ABB RobotStudio station: Session5.rspag

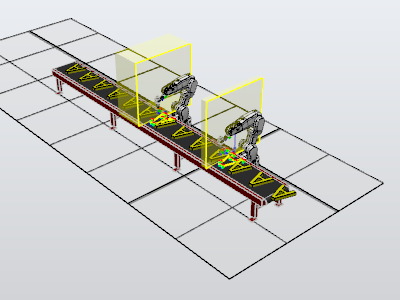
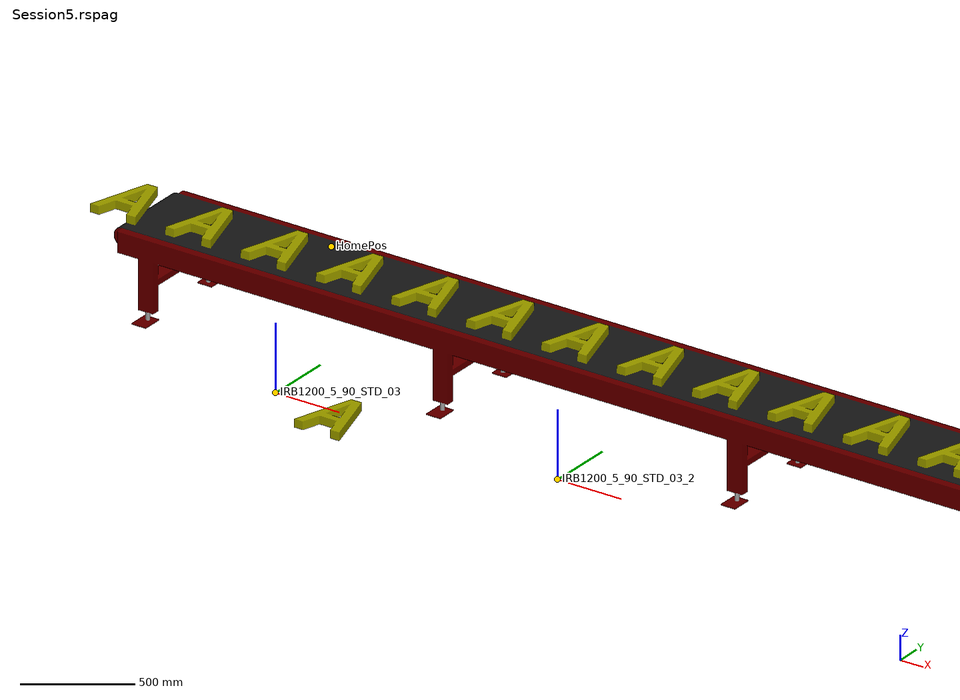
[picture v1: parts stored in the station drawn from their meshes, with robot base, taught points and paths (robot models come from the ABB library and are not in the file)]
--- station ---
Station Session5 (saved by RobotStudio 24.2.10821.1)
Controller IRB1200_CNV_2, task T_ROB1: task frame (RAPID world) sits at (1000, 521.42, 400) mm in the station
Controller IRB1200_CNV_1, task T_ROB1: task frame (RAPID world) sits at (-500, 521.42, 400) mm in the station
Controller IRB1200_CNV_1
  mechanical unit ROB_1: IRB1200_5_90_STD_03, 6 joints, base frame (0, -290, -400) mm, rotated rx 0 ry 0 rz 90 deg
  mechanical unit CNV1: ?, 1 joints, base frame (0, 0, 0) mm
Controller IRB1200_CNV_2
  mechanical unit ROB_1: IRB1200_5_90_STD_03_2, 6 joints, base frame (0, -290, -400) mm, rotated rx 0 ry 0 rz 90 deg
  mechanical unit CNV1: ?, 1 joints, base frame (0, 0, 0) mm
Layout (positions relative to the parent item):
  - IRB1200_5_90_STD_03 [mechanism, from %ABB.RobotStudio.Models.IRB1200%\IRB1200_5_90_STD_03.rslib] at (-500, 231.42, 0) mm, rotated rx 0 ry 0 rz 90 deg; joint values [-0.0648, -0.2584, 0.4127, -0.0339, 0.7666, 0.0529] (rad or m)
  - mySpintecTool [mechanism, from Library\mySpintecTool.rslib] at (-472.99, 617.74, 739.17) mm, rotated rx -179.89 ry 37.27 rz -95.76 deg
  - Conveyor 1 [conveyor]
    - Belt Conveyor [part] at (-518.08, 731.42, 0) mm, size 5091 x 600 x 400 mm
    - Product_A [part], size 239 x 301.5 x 40 mm
    - ConveyorObject_82 [conveyorobject] at (3315.13, 521.42, 400) mm
      - Product_A [part] at (0, 50, 0) mm, size 239 x 301.5 x 40 mm
    - ConveyorObject_83 [conveyorobject] at (2915.13, 521.42, 400) mm
      - Product_A [part] at (0, 50, 0) mm, size 239 x 301.5 x 40 mm
    - ConveyorObject_84 [conveyorobject] at (2515.13, 521.42, 400) mm
      - Product_A [part] at (0, 50, 0) mm, size 239 x 301.5 x 40 mm
    - ConveyorObject_85 [conveyorobject] at (2115.13, 521.42, 400) mm
      - Product_A [part] at (0, 50, 0) mm, size 239 x 301.5 x 40 mm
    - ConveyorObject_86 [conveyorobject] at (1715.13, 521.42, 400) mm
      - Product_A [part] at (0, 50, 0) mm, size 239 x 301.5 x 40 mm
    - ConveyorObject_87 [conveyorobject] at (1315.13, 521.42, 400) mm
      - Product_A [part] at (0, 50, 0) mm, size 239 x 301.5 x 40 mm
    - ConveyorObject_88 [conveyorobject] at (915.13, 521.42, 400) mm
      - Product_A [part] at (0, 50, 0) mm, size 239 x 301.5 x 40 mm
    - ConveyorObject_89 [conveyorobject] at (515.13, 521.42, 400) mm
      - Product_A [part] at (0, 50, 0) mm, size 239 x 301.5 x 40 mm
    - ConveyorObject_90 [conveyorobject] at (115.13, 521.42, 400) mm
      - Product_A [part] at (0, 50, 0) mm, size 239 x 301.5 x 40 mm
    - ConveyorObject_91 [conveyorobject] at (-284.87, 521.42, 400) mm
      - Product_A [part] at (0, 50, 0) mm, size 239 x 301.5 x 40 mm
    - ConveyorObject_92 [conveyorobject] at (-684.87, 521.42, 400) mm
      - Product_A [part] at (0, 50, 0) mm, size 239 x 301.5 x 40 mm
    - ConveyorObject_93 [conveyorobject] at (-1084.87, 521.42, 400) mm
      - Product_A [part] at (0, 50, 0) mm, size 239 x 301.5 x 40 mm
    - ConveyorObject_94 [conveyorobject] at (-1484.87, 521.42, 400) mm
      - Product_A [part] at (0, 50, 0) mm, size 239 x 301.5 x 40 mm
  - IRB1200_5_90_STD_03_2 [mechanism, from %ABB.RobotStudio.Models.IRB1200%\IRB1200_5_90_STD_03.rslib] at (1000, 231.42, 0) mm, rotated rx 0 ry 0 rz 90 deg; joint values [0, -0.4363, 0.5236, 0, 0.8378, 0] (rad or m)
  - mySpintecTool_2 [mechanism, from Library\mySpintecTool.rslib] at (1000, 544.38, 742.17) mm, rotated rx 180 ry 37 rz -90 deg
Attachment: mySpintecTool is attached to IRB1200_5_90_STD_03 / Link6
Attachment: mySpintecTool_2 is attached to IRB1200_5_90_STD_03_2 / Link6
Conveyor tracking Connection: unit CNV1, TravelOffset=1.018075, QueueTrackDistance=0, StartWindowWidth=0.1, SyncSeparation=5E-06, CountsPerMeter=20000
Conveyor tracking Connection_2: unit CNV1, TravelOffset=2.518075, QueueTrackDistance=0, StartWindowWidth=0.5, SyncSeparation=5E-06, CountsPerMeter=20000
Targets, tools, work objects and paths stored in the station and not in the controller backup, written as RAPID:
! task T_ROB1
MODULE Module1
  CONST robtarget Target_10:=[[0,50,40],[0,-0.595435711,0.803402959,0],[0,0,0,0],[9E+09,9E+09,9E+09,9E+09,9E+09,0]];
ENDMODULE


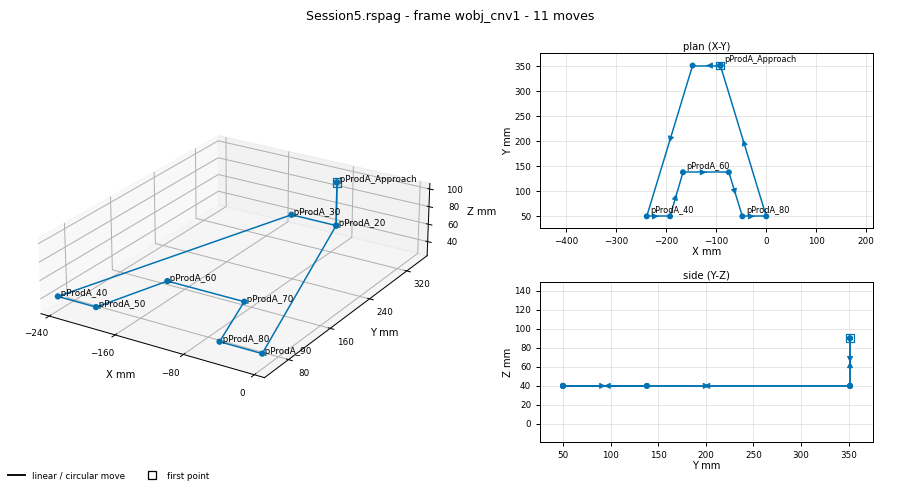
[picture p0: tool path of Session5.rspag in frame wobj_cnv1, 11 of 13 moves have a stored position in this frame; points joined in program order, loops and branches not executed]
--- Backups/IRB1200_CNV_1/RAPID/TASK1/PROGMOD/CalibData.mod ---
MODULE CalibData
    PERS tooldata tSpintec:=[TRUE,[[31.792631019,0,229.638935148],[0.945518576,0,0.325568154,0]],[3,[-51.132047978,0,99.657990242],[1,0,0,0],0,0,0]];
    TASK PERS wobjdata wobj_cnv1:=[FALSE,FALSE,"CNV1",[[0,0,0],[1,0,0,0]],[[0,0,0],[1,0,0,0]]];
ENDMODULE

--- Backups/IRB1200_CNV_1/RAPID/TASK1/PROGMOD/Module1.mod ---
MODULE Module1
        CONST robtarget pProdA_Approach:=[[-91.678309329,351.549379803,90],[0,-0.595435711,0.803402959,0],[0,-1,0,0],[9E+09,9E+09,9E+09,9E+09,9E+09,0]];
    CONST robtarget pProdA_20:=[[-91.678309329,351.549379803,40],[0,-0.595435711,0.803402959,0],[0,-1,0,0],[9E+09,9E+09,9E+09,9E+09,9E+09,0]];
    CONST robtarget pProdA_30:=[[-147.312155161,351.549379803,40],[0,-0.595435711,0.803402959,0],[0,-1,0,0],[9E+09,9E+09,9E+09,9E+09,9E+09,0]];
    CONST robtarget pProdA_40:=[[-239.002311678,50,40],[0,-0.595435711,0.803402959,0],[0,-1,1,0],[9E+09,9E+09,9E+09,9E+09,9E+09,0]];
    CONST robtarget pProdA_50:=[[-192.367734531,50,40],[0,-0.595435711,0.803402959,0],[0,-1,0,0],[9E+09,9E+09,9E+09,9E+09,9E+09,0]];
    CONST robtarget pProdA_60:=[[-166.509749849,138.164676665,40],[0,-0.595435711,0.803402959,0],[0,-1,0,0],[9E+09,9E+09,9E+09,9E+09,9E+09,0]];
    CONST robtarget pProdA_70:=[[-74.83144052,138.164676665,40],[0,-0.595435711,0.803402959,0],[0,-1,0,0],[9E+09,9E+09,9E+09,9E+09,9E+09,0]];
    CONST robtarget pProdA_80:=[[-47.798092898,50,40],[0,-0.595435711,0.803402959,0],[0,-1,0,0],[9E+09,9E+09,9E+09,9E+09,9E+09,0]];
    CONST robtarget pProdA_90:=[[0,50,40],[0,-0.595435711,0.803402959,0],[0,-1,0,0],[9E+09,9E+09,9E+09,9E+09,9E+09,0]];
    CONST robtarget HomePos:=[[0,135.769637657,139.639623038],[0.006170592,0.707079857,-0.707079857,0.006170592],[0,0,0,0],[9E+09,9E+09,9E+09,9E+09,9E+09,0]];
!***********************************************************
    !
    ! Module:  Module1
    !
    ! Description:
    !   <Insert description here>
    !
    ! Author: ahmadk
    !
    ! Version: 1.0
    !
    !***********************************************************


    !***********************************************************
    !
    ! Procedure main
    !
    !   This is the entry point of your program
    !
    !***********************************************************
    PROC main()
        !Add your code here
        MoveJ HomePos,v5000,fine,tSpintec\WObj:=wobj0;
        ActUnit CNV1;
        Confl \Off;
        WHILE TRUE DO
            WaitWObj wobj_cnv1;
            Product_A;
            MoveJ HomePos,v5000,fine,tSpintec\WObj:=wobj0;
            DropWObj wobj_cnv1;
        ENDWHILE

    ENDPROC
    PROC Product_A()
        MoveL pProdA_Approach,v500,z1,tSpintec\WObj:=wobj_cnv1;
        MoveL pProdA_20,v500,z1,tSpintec\WObj:=wobj_cnv1;
        MoveL pProdA_30,v500,z1,tSpintec\WObj:=wobj_cnv1;
        MoveL pProdA_40,v500,z1,tSpintec\WObj:=wobj_cnv1;
        MoveL pProdA_50,v500,z1,tSpintec\WObj:=wobj_cnv1;
        MoveL pProdA_60,v500,z1,tSpintec\WObj:=wobj_cnv1;
        MoveL pProdA_70,v500,z1,tSpintec\WObj:=wobj_cnv1;
        MoveL pProdA_80,v500,z1,tSpintec\WObj:=wobj_cnv1;
        MoveL pProdA_90,v500,z1,tSpintec\WObj:=wobj_cnv1;
        MoveL pProdA_20,v500,z1,tSpintec\WObj:=wobj_cnv1;
        MoveL pProdA_Approach,v500,z1,tSpintec\WObj:=wobj_cnv1;
    ENDPROC
ENDMODULE

--- Backups/IRB1200_CNV_1/SYSPAR/EIO.cfg ---
EIO:CFG_1.0:6:1::
#
INDUSTRIAL_NETWORK:

      -Name "DeviceNet" -Label "DeviceNet Master/Slave Network" -Address "2"
#
DEVICENET_DEVICE:

      -Name "Qtrack1" -Simulated  -VendorName "ABB Robotics"\
      -ProductName "Qtracker" -Address 15 -ProductCode 16 -DeviceType 100\
      -PollRate 20 -OutputSize 6 -InputSize 19
#
DEVICENET_DEVICE_TEMPLATE:

      -Name "d377B" -VendorName "ABB Robotics" -ProductName "Qtracker"\
      -Label "DSQC 377B Queue Tracker" -ProductCode 16 -DeviceType 100\
      -PollRate 20 -OutputSize 6 -InputSize 19
#
DEVICENET_COMMAND:

      -Name "CountsPerMeter1" -Device "Qtrack1" -OrderNr 2\
      -Path "6,20 66 24 01 30 01,CA,4" -Value "20000"

      -Name "SyncSeparation1" -Device "Qtrack1" -OrderNr 3\
      -Path "6,20 66 24 01 30 02,CA,4" -Value "0.005"

      -Name "QueueTrckDist1" -Device "Qtrack1" -OrderNr 4\
      -Path "6,20 66 24 01 30 03,CA,4" -Value "0"

      -Name "StartWinWidth1" -Device "Qtrack1" -OrderNr 5\
      -Path "6,20 66 24 01 30 04,CA,4" -Value "100"

      -Name "AutoBackup1" -Device "Qtrack1" -OrderNr 6\
      -Path "6,20 66 24 01 30 12,C1,1" -Value "1"

      -Name "SimulationVel1" -Device "Qtrack1" -OrderNr 7\
      -Path "6,20 66 24 01 30 13,CA,4" -Value "0.100"

      -Name "ScalingFactor1" -Device "Qtrack1" -OrderNr 8\
      -Path "6,20 66 24 01 30 14,CA,4" -Value "2000.0"

      -Name "CheckPointDist1" -Device "Qtrack1" -OrderNr 9\
      -Path "6,20 66 24 01 30 15,CA,4" -Value "0.0"

      -Name "CheckPWinWidth1" -Device "Qtrack1" -OrderNr 10\
      -Path "6,20 66 24 01 30 16,CA,4" -Value "0.0"

      -Name "IIRFPeriod1" -Device "Qtrack1" -OrderNr 11\
      -Path "6,20 66 24 01 30 05,CA,4" -Value "0.02"

      -Name "IIRFNoOfPoles1" -Device "Qtrack1" -OrderNr 12\
      -Path "6,20 66 24 01 30 06,C6,1" -Value "2"

      -Name "IIRFNoOfZeroes1" -Device "Qtrack1" -OrderNr 13\
      -Path "6,20 66 24 01 30 07,C6,1" -Value "0"

      -Name "IIRFXfrmMetPol1" -Device "Qtrack1" -OrderNr 14\
      -Path "6,20 66 24 01 30 08,C6,1" -Value "1"

      -Name "IIRFXfrmMetZero1" -Device "Qtrack1" -OrderNr 15\
      -Path "6,20 66 24 01 30 09,C6,1" -Value "1"

      -Name "IIRFFZ1" -Device "Qtrack1" -OrderNr 16\
      -Path "6,20 66 24 01 30 0A,CA,4" -Value "0.0"

      -Name "IIRFDZ1" -Device "Qtrack1" -OrderNr 17\
      -Path "6,20 66 24 01 30 0B,CA,4" -Value "0.0"

      -Name "IIRFFP1" -Device "Qtrack1" -OrderNr 18\
      -Path "6,20 66 24 01 30 0C,CA,4" -Value "2.0"

      -Name "IIRFDP1" -Device "Qtrack1" -OrderNr 19\
      -Path "6,20 66 24 01 30 0D,CA,4" -Value "0.707"

      -Name "IIRFGain1" -Device "Qtrack1" -OrderNr 20\
      -Path "6,20 66 24 01 30 0E,CA,4" -Value "1.0"

      -Name "FIRFLength1" -Device "Qtrack1" -OrderNr 21\
      -Path "6,20 66 24 01 30 0F,C6,1" -Value "0"

      -Name "FIRFB01" -Device "Qtrack1" -OrderNr 22\
      -Path "6,20 66 24 01 30 10,CA,4" -Value "0.0"

      -Name "FIRFB11" -Device "Qtrack1" -OrderNr 23\
      -Path "6,20 66 24 01 30 11,CA,4" -Value "0.0"
#
DEVICENET_INTERNAL_DEVICE:

      -Name "DN_Internal_Device" -VendorName "ABB Robotics"\
      -ProductName "DeviceNet Internal Slave Device"
#
EIO_SIGNAL:

      -Name "c1Position" -SignalType "AI" -Device "Qtrack1" -DeviceMap "0-31"\
      -MaxLog 21474.8 -MaxPhys 1 -MaxPhysLimit 1 -MaxBitVal 2147483647\
      -MinLog -21474.8 -MinPhys -1 -MinPhysLimit -1 -MinBitVal -2147483647

      -Name "c1Speed" -SignalType "AI" -Device "Qtrack1" -DeviceMap "32-63"\
      -MaxLog 21474.8 -MaxPhys 1 -MaxPhysLimit 1 -MaxBitVal 2147483647\
      -MinLog -21474.8 -MinPhys -1 -MinPhysLimit -1 -MinBitVal -2147483647

      -Name "c1Connected" -SignalType "DI" -Device "Qtrack1" -DeviceMap "104"

      -Name "c1NullSpeed" -SignalType "DI" -Device "Qtrack1" -DeviceMap "105"

      -Name "c1DReady" -SignalType "DI" -Device "Qtrack1" -DeviceMap "106"

      -Name "c1PassStw" -SignalType "DI" -Device "Qtrack1" -DeviceMap "107"

      -Name "c1NewObjStrobe" -SignalType "DI" -Device "Qtrack1" -DeviceMap "108"

      -Name "c1EncSelected" -SignalType "DI" -Device "Qtrack1" -DeviceMap "109"

      -Name "c1EncAFautlt" -SignalType "DI" -Device "Qtrack1" -DeviceMap "110"

      -Name "c1EncBFautlt" -SignalType "DI" -Device "Qtrack1" -DeviceMap "111"

      -Name "c1Simulating" -SignalType "DI" -Device "Qtrack1" -DeviceMap "112"

      -Name "c1DirOfTravel" -SignalType "DI" -Device "Qtrack1" -DeviceMap "113"

      -Name "c1ScaleEncPuls" -SignalType "DI" -Device "Qtrack1" -DeviceMap "114"

      -Name "c1PowerUpStatus" -SignalType "DI" -Device "Qtrack1" -DeviceMap "83"

      -Name "c1WaitWObj" -SignalType "DO" -Device "Qtrack1" -DeviceMap "0"

      -Name "c1DropWObj" -SignalType "DO" -Device "Qtrack1" -DeviceMap "1"

      -Name "c1Rem1PObj" -SignalType "DO" -Device "Qtrack1" -DeviceMap "2"

      -Name "c1RemAllPObj" -SignalType "DO" -Device "Qtrack1" -DeviceMap "3"

      -Name "c1EncSelect" -SignalType "DO" -Device "Qtrack1" -DeviceMap "4"

      -Name "c1SoftSyncSig" -SignalType "DO" -Device "Qtrack1" -DeviceMap "5"

      -Name "c1SoftCheckSig" -SignalType "DO" -Device "Qtrack1" -DeviceMap "6"

      -Name "c1SimMode" -SignalType "DO" -Device "Qtrack1" -DeviceMap "7"

      -Name "c1CntToEncStr" -SignalType "DO" -Device "Qtrack1" -DeviceMap "40"

      -Name "c1ForceJob" -SignalType "DO" -Device "Qtrack1" -DeviceMap "41"

      -Name "c1PosInJobQ" -SignalType "DO" -Device "Qtrack1" -DeviceMap "42"

      -Name "c1ObjectsInQ" -SignalType "GI" -Device "Qtrack1" -DeviceMap "64-71"

      -Name "c1CntFromEnc" -SignalType "GI" -Device "Qtrack1"\
      -DeviceMap "72-103"

      -Name "c1DTimestamp" -SignalType "GI" -Device "Qtrack1"\
      -DeviceMap "120-151"

      -Name "c1CntToEnc" -SignalType "GO" -Device "Qtrack1" -DeviceMap "8-39"

--- Backups/IRB1200_CNV_1/SYSPAR/PROC.cfg ---
PROC:CFG_1.0:6:0::
#
CONVEYOR:

      -name "CNV1" -sensor_type "CAN" -use_sensor "CAN1" -adjustment_speed 850\
      -min_dist -600 -max_dist 20000 -correction_vector_ramp_length 5
#
CONVEYOR_CAN_SENSOR:

      -name "CAN1" -eio_unit_name "Qtrack1" -connected_signal "c1Connected"\
      -position_signal "c1Position" -velocity_signal "c1Speed"\
      -null_speed_signal "c1NullSpeed" -wait_wobj_signal "c1WaitWObj"\
      -drop_wobj_signal "c1DropWObj" -data_timestamp "c1DTimestamp"\
      -rem_all_pobj_signal "c1RemAllPObj" -rem_one_pobj_signal "c1Rem1PObj"\
      -supervise_max_dist_off  -newobj_strobe "c1NewObjStrobe"\
      -encA_fault_signal "c1EncAFautlt" -dir_of_travel_signal "c1DirOfTravel"\
      -force_job_signal "c1ForceJob" -count_to_enc_strobe "c1CntToEncStr"\
      -pos_in_jobq_signal "c1PosInJobQ" -obj_in_queue_signal "c1ObjectsInQ"\
      -count_from_enc "c1CntFromEnc" -count_to_enc "c1CntToEnc"\
      -scale_enc_puls "c1ScaleEncPuls"

--- Backups/IRB1200_CNV_2/SYSPAR/EIO.cfg ---
EIO:CFG_1.0:6:1::
#
INDUSTRIAL_NETWORK:

      -Name "DeviceNet" -Label "DeviceNet Master/Slave Network" -Address "2"
#
DEVICENET_DEVICE:

      -Name "Qtrack1" -Simulated  -VendorName "ABB Robotics"\
      -ProductName "Qtracker" -Address 15 -ProductCode 16 -DeviceType 100\
      -PollRate 20 -OutputSize 6 -InputSize 19
#
DEVICENET_DEVICE_TEMPLATE:

      -Name "d377B" -VendorName "ABB Robotics" -ProductName "Qtracker"\
      -Label "DSQC 377B Queue Tracker" -ProductCode 16 -DeviceType 100\
      -PollRate 20 -OutputSize 6 -InputSize 19
#
DEVICENET_COMMAND:

      -Name "CountsPerMeter1" -Device "Qtrack1" -OrderNr 2\
      -Path "6,20 66 24 01 30 01,CA,4" -Value "20000"

      -Name "SyncSeparation1" -Device "Qtrack1" -OrderNr 3\
      -Path "6,20 66 24 01 30 02,CA,4" -Value "0.005"

      -Name "QueueTrckDist1" -Device "Qtrack1" -OrderNr 4\
      -Path "6,20 66 24 01 30 03,CA,4" -Value "0"

      -Name "StartWinWidth1" -Device "Qtrack1" -OrderNr 5\
      -Path "6,20 66 24 01 30 04,CA,4" -Value "500"

      -Name "AutoBackup1" -Device "Qtrack1" -OrderNr 6\
      -Path "6,20 66 24 01 30 12,C1,1" -Value "1"

      -Name "SimulationVel1" -Device "Qtrack1" -OrderNr 7\
      -Path "6,20 66 24 01 30 13,CA,4" -Value "0.100"

      -Name "ScalingFactor1" -Device "Qtrack1" -OrderNr 8\
      -Path "6,20 66 24 01 30 14,CA,4" -Value "2000.0"

      -Name "CheckPointDist1" -Device "Qtrack1" -OrderNr 9\
      -Path "6,20 66 24 01 30 15,CA,4" -Value "0.0"

      -Name "CheckPWinWidth1" -Device "Qtrack1" -OrderNr 10\
      -Path "6,20 66 24 01 30 16,CA,4" -Value "0.0"

      -Name "IIRFPeriod1" -Device "Qtrack1" -OrderNr 11\
      -Path "6,20 66 24 01 30 05,CA,4" -Value "0.02"

      -Name "IIRFNoOfPoles1" -Device "Qtrack1" -OrderNr 12\
      -Path "6,20 66 24 01 30 06,C6,1" -Value "2"

      -Name "IIRFNoOfZeroes1" -Device "Qtrack1" -OrderNr 13\
      -Path "6,20 66 24 01 30 07,C6,1" -Value "0"

      -Name "IIRFXfrmMetPol1" -Device "Qtrack1" -OrderNr 14\
      -Path "6,20 66 24 01 30 08,C6,1" -Value "1"

      -Name "IIRFXfrmMetZero1" -Device "Qtrack1" -OrderNr 15\
      -Path "6,20 66 24 01 30 09,C6,1" -Value "1"

      -Name "IIRFFZ1" -Device "Qtrack1" -OrderNr 16\
      -Path "6,20 66 24 01 30 0A,CA,4" -Value "0.0"

      -Name "IIRFDZ1" -Device "Qtrack1" -OrderNr 17\
      -Path "6,20 66 24 01 30 0B,CA,4" -Value "0.0"

      -Name "IIRFFP1" -Device "Qtrack1" -OrderNr 18\
      -Path "6,20 66 24 01 30 0C,CA,4" -Value "2.0"

      -Name "IIRFDP1" -Device "Qtrack1" -OrderNr 19\
      -Path "6,20 66 24 01 30 0D,CA,4" -Value "0.707"

      -Name "IIRFGain1" -Device "Qtrack1" -OrderNr 20\
      -Path "6,20 66 24 01 30 0E,CA,4" -Value "1.0"

      -Name "FIRFLength1" -Device "Qtrack1" -OrderNr 21\
      -Path "6,20 66 24 01 30 0F,C6,1" -Value "0"

      -Name "FIRFB01" -Device "Qtrack1" -OrderNr 22\
      -Path "6,20 66 24 01 30 10,CA,4" -Value "0.0"

      -Name "FIRFB11" -Device "Qtrack1" -OrderNr 23\
      -Path "6,20 66 24 01 30 11,CA,4" -Value "0.0"
#
DEVICENET_INTERNAL_DEVICE:

      -Name "DN_Internal_Device" -VendorName "ABB Robotics"\
      -ProductName "DeviceNet Internal Slave Device"
#
EIO_SIGNAL:

      -Name "c1Position" -SignalType "AI" -Device "Qtrack1" -DeviceMap "0-31"\
      -MaxLog 21474.8 -MaxPhys 1 -MaxPhysLimit 1 -MaxBitVal 2147483647\
      -MinLog -21474.8 -MinPhys -1 -MinPhysLimit -1 -MinBitVal -2147483647

      -Name "c1Speed" -SignalType "AI" -Device "Qtrack1" -DeviceMap "32-63"\
      -MaxLog 21474.8 -MaxPhys 1 -MaxPhysLimit 1 -MaxBitVal 2147483647\
      -MinLog -21474.8 -MinPhys -1 -MinPhysLimit -1 -MinBitVal -2147483647

      -Name "c1Connected" -SignalType "DI" -Device "Qtrack1" -DeviceMap "104"

      -Name "c1NullSpeed" -SignalType "DI" -Device "Qtrack1" -DeviceMap "105"

      -Name "c1DReady" -SignalType "DI" -Device "Qtrack1" -DeviceMap "106"

      -Name "c1PassStw" -SignalType "DI" -Device "Qtrack1" -DeviceMap "107"

      -Name "c1NewObjStrobe" -SignalType "DI" -Device "Qtrack1" -DeviceMap "108"

      -Name "c1EncSelected" -SignalType "DI" -Device "Qtrack1" -DeviceMap "109"

      -Name "c1EncAFautlt" -SignalType "DI" -Device "Qtrack1" -DeviceMap "110"

      -Name "c1EncBFautlt" -SignalType "DI" -Device "Qtrack1" -DeviceMap "111"

      -Name "c1Simulating" -SignalType "DI" -Device "Qtrack1" -DeviceMap "112"

      -Name "c1DirOfTravel" -SignalType "DI" -Device "Qtrack1" -DeviceMap "113"

      -Name "c1ScaleEncPuls" -SignalType "DI" -Device "Qtrack1" -DeviceMap "114"

      -Name "c1PowerUpStatus" -SignalType "DI" -Device "Qtrack1" -DeviceMap "83"

      -Name "c1WaitWObj" -SignalType "DO" -Device "Qtrack1" -DeviceMap "0"

      -Name "c1DropWObj" -SignalType "DO" -Device "Qtrack1" -DeviceMap "1"

      -Name "c1Rem1PObj" -SignalType "DO" -Device "Qtrack1" -DeviceMap "2"

      -Name "c1RemAllPObj" -SignalType "DO" -Device "Qtrack1" -DeviceMap "3"

      -Name "c1EncSelect" -SignalType "DO" -Device "Qtrack1" -DeviceMap "4"

      -Name "c1SoftSyncSig" -SignalType "DO" -Device "Qtrack1" -DeviceMap "5"

      -Name "c1SoftCheckSig" -SignalType "DO" -Device "Qtrack1" -DeviceMap "6"

      -Name "c1SimMode" -SignalType "DO" -Device "Qtrack1" -DeviceMap "7"

      -Name "c1CntToEncStr" -SignalType "DO" -Device "Qtrack1" -DeviceMap "40"

      -Name "c1ForceJob" -SignalType "DO" -Device "Qtrack1" -DeviceMap "41"

      -Name "c1PosInJobQ" -SignalType "DO" -Device "Qtrack1" -DeviceMap "42"

      -Name "c1ObjectsInQ" -SignalType "GI" -Device "Qtrack1" -DeviceMap "64-71"

      -Name "c1CntFromEnc" -SignalType "GI" -Device "Qtrack1"\
      -DeviceMap "72-103"

      -Name "c1DTimestamp" -SignalType "GI" -Device "Qtrack1"\
      -DeviceMap "120-151"

      -Name "c1CntToEnc" -SignalType "GO" -Device "Qtrack1" -DeviceMap "8-39"
